VAR_GLOBAL
	stackerCraneProcess : StackerCraneProcess;
END_VAR

(* stored: Version 1.1.0.1, ProductVersion 3.1.4024.10
   GVL GVL_Processes: Id {14ac167a-9928-460c-a0e3-530eb8b69a9b} *)
